(* Schneider Machine Expert - Basic project p11, file version 1.8.0.0 *)
(* ProjectInformations: Name=New project *)

HARDWARE
  Cpu 0: TM221CE16R
  EthernetConfiguration: NetworkName=M221, IpAllocationMode=FixedAddress, IpAddress=192.168.162.202, SubnetMask=255.255.255.0
  SerialLineConfiguration: Baud=Baud19200, Parity=ParityEven, DataBits=DataBits8, StopBits=StopBits1, PhysicalMedium=PhysicalMediumRs485, TransmissionMode=TransmissionModeModbusRtu, SlaveId=1, Addressing=SlaveAddressing
  MastTask: UsePeriodScanMode=false, PeriodScan=100
  FastTask: Period=255
  CpuBehavior: StartingMode=StartAsPreviousState, AutoSaveRamOnEeprom=true, WatchdogPeriod=250

SYMBOLS  (address, symbol, comment, settings)
  %TM0        [Preset=1, Base=OneSecond, IsRetentive=true]
  %TM1        [Preset=1, Base=OneSecond, IsRetentive=true]

POU New POU
  (* SectionNumber=1 *)

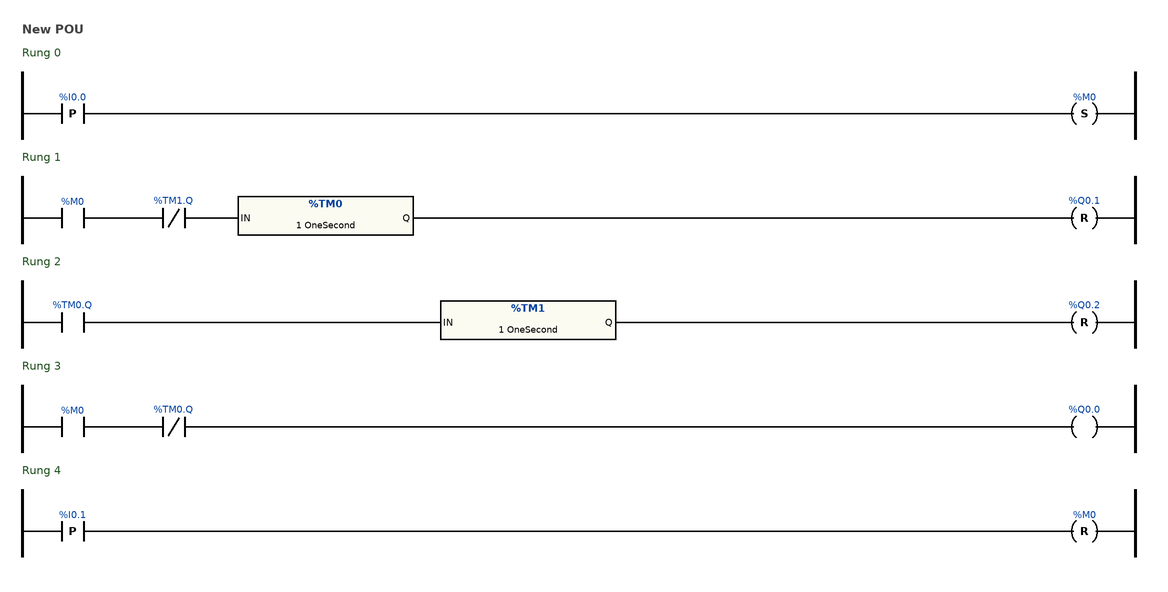

// Rung 0
  LDR %I0.0
  S %M0
  // as ST:
  //   IF RISING(%I0.0) THEN %M0 := TRUE; END_IF;

// Rung 1
  BLK %TM0
  LD %M0
  ANDN %TM1.Q
  IN
  OUT_BLK
  LD Q
  R %Q0.1
  END_BLK
  // as ST:
  //   %TM0(IN := %M0 AND NOT %TM1.Q);
  //   IF %TM0.Q THEN %Q0.1 := FALSE; END_IF;

// Rung 2
  BLK %TM1
  LD %TM0.Q
  IN
  OUT_BLK
  LD Q
  R %Q0.2
  END_BLK
  // as ST:
  //   %TM1(IN := %TM0.Q);
  //   IF %TM1.Q THEN %Q0.2 := FALSE; END_IF;

// Rung 3
  LD %M0
  ANDN %TM0.Q
  ST %Q0.0
  // as ST:
  //   %Q0.0 := %M0 AND NOT %TM0.Q;

// Rung 4
  LDR %I0.1
  R %M0
  // as ST:
  //   IF RISING(%I0.1) THEN %M0 := FALSE; END_IF;
